SUBAPPLICATION ObjectPointer_Swap_AX (* Schaltet einen ObjectPointer (CPointer) bei DI1=TRUE auf u16ObjId_Show um, bei FALSE auf ID_NULL (nichts sichtbar). ISO 11783-6 F.22 'Change Numeric Value' (Q_NumericValue) - ObjectPointer liegt explizit in dessen gueltigem Object-ID-Bereich (27000-27999). NICHT F.38 'Change Attribute' (Q_Attribute) verwenden - AID_OP_PTR.VALUE ist dort read-only. Muster: ms-train/4diac_training1 Ventilsteuerung/4diacIDE-workspace/test_B/Uebungen/Uebung_015.SUB (Franz). *)
  (* Standard: 61499-2; Description: Copyright (c) 2026 Meisterschulen am Ostbahnhof This program and the accompanying materials are made available under the terms of the Eclipse Public License 2.0 which is available at https://www.eclipse.org/legal/epl-2.0/ SPDX-License-Identifier: EPL-2.0 *)
  (* Version 1.0, 2026-09-29, Franz Höpfinger, Meisterschulen am Ostbahnhof, initial implementation, analog GreenWhiteBackground1_AX (AX_SEL-Wrapper um eine Q_-FB) - Franz-Korrektur: Q_Attribute/F.38 verworfen, Q_NumericValue/F.22 ist der richtige Weg fuer ObjectPointer. *)
  PACKAGE MyLib::sys;
  IMPORT isobus::UT::Q::const::IDs::ID_NULL;
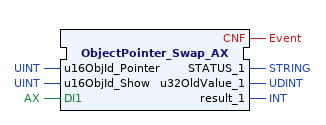
  EVENT_OUTPUT
    CNF; (* Execution Confirmation *)
  END_EVENT
  VAR_INPUT
    u16ObjId_Pointer : UINT := ID_NULL; (* Object ID des ObjectPointer (CPointer), dessen Ziel geschaltet wird *)
    u16ObjId_Show : UINT := ID_NULL; (* Object ID, die bei DI1=TRUE unter dem Pointer angezeigt wird *)
  END_VAR
  VAR_OUTPUT
    STATUS_1 : STRING; (* Service Status *)
    u32OldValue_1 : UDINT; (* Old value of ID *)
    result_1 : INT; (* retval see description *)
  END_VAR
  SOCKETS
    DI1 : adapter::types::unidirectional::AX; (* Selector *)
  END_SOCKETS
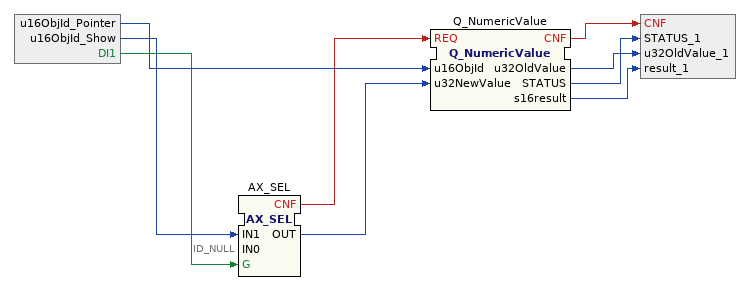
  FBS
    Q_NumericValue : isobus::UT::Q::Q_NumericValue;
    AX_SEL : adapter::iec61131::selection::AX_SEL(IN0 := ID_NULL);
  END_FBS
  EVENT_CONNECTIONS
    Q_NumericValue.CNF TO CNF;
    AX_SEL.CNF TO Q_NumericValue.REQ;
  END_CONNECTIONS
  DATA_CONNECTIONS
    u16ObjId_Pointer TO Q_NumericValue.u16ObjId;
    u16ObjId_Show TO AX_SEL.IN1;
    Q_NumericValue.u32OldValue TO u32OldValue_1;
    Q_NumericValue.STATUS TO STATUS_1;
    Q_NumericValue.s16result TO result_1;
    AX_SEL.OUT TO Q_NumericValue.u32NewValue;
  END_CONNECTIONS
  ADAPTER_CONNECTIONS
    DI1 TO AX_SEL.G;
  END_CONNECTIONS
END_SUBAPPLICATION
